PROGRAM PRG_Com
VAR
	i :INT;
END_VAR

METHOD M_Add : BOOL
VAR_INPUT
END_VAR
i:=i+1;
END_METHOD

END_PROGRAM

(* stored: Version 1.1.0.1, ProductVersion 3.1.4024.2
   POU PRG_Com: Id {230547be-281f-45f8-b65d-c19832a9bfb9}, SpecialFunc None
   Method M_Add: Id {45c06027-5a71-4197-9ae6-90436419f4a7} *)
